{attribute addProperty BoxType "EL5001--0000"}
{attribute addProperty Id "StatusAT %I*BYTE811ValueAT %I*UDINT3242"}
{attribute addProperty CRC "1947596278"}
{attribute addProperty SizeInBites "40"}
{attribute addProperty SizeInBytes "5"}
TYPE Channel_7415F5F6 :
STRUCT
	{attribute addProperty Name "Status"}
	Status AT %I* : BYTE;
	{attribute addProperty Name "Value"}
	Value AT %I* : UDINT;
END_STRUCT
END_TYPE

(* stored: Version 1.2.0.0, ProductVersion 3.1.4024.9
   DUT Channel_7415F5F6: Id {3bd54a3d-65b6-47e1-93fe-2365d67f79c5} *)
